(* IEC 61131-3 sources: programs/VI-54/VI-54_20171205/VI-54_20171205/Stations/PLC_VI54/VI-54_171014/Class/Claxon, 1 file *)

(* ---- Claxon.st ---- *)
(*!
<Class
	Name               = "Claxon"
	Revision           = "0.0"
	RealtimeTask       = "false"
	CyclicTask         = "false"
	BackgroundTask     = "false"
	Sigmatek           = "false"
	OSInterface        = "false"
	HighPriority       = "false"
	Automatic          = "false"
	UpdateMode         = "Prescan"
	SharedCommandTable = "true"
	Objectsize         = "(480,120)">
	<Channels>
		<Server Name="ClaxonActief" Visualized="true" Initialize="true" WriteProtected="false" Retentive="false"/>
		<Server Name="Comm" Visualized="false" Initialize="false" WriteProtected="true" Retentive="false"/>
		<Client Name="oClaxon" Required="false" Internal="false"/>
	</Channels>
</Class>
*)
Claxon : CLASS
  //Servers:
	Comm 	: SvrChCmd_DINT;
	ClaxonActief 	: SvrCh_OptiesEnum;
  //Clients:
	oClaxon 	: CltCh_DINT;
  //Variables:
  //Functions:

	FUNCTION GLOBAL ClaxonState
		VAR_INPUT
			State 	: DINT;
		END_VAR;
  //Tables:
	FUNCTION @STD
		VAR_OUTPUT
			ret_code	: CONFSTATES;
		END_VAR;
	FUNCTION GLOBAL TAB @CT_;
END_CLASS;

FUNCTION GLOBAL Claxon::ClaxonState
	VAR_INPUT
		State 	: DINT;
	END_VAR

  if ClaxonActief = Actief then
    oClaxon := State;
  else
    oClaxon := 0;
  end_if;

  oClaxon.Write(input:= oClaxon);

END_FUNCTION
